{attribute 'qualified_only'}
VAR_GLOBAL CONSTANT
    nNumberOfFilterConstantThicknessSlotsInHolder : INT := 11;
    nNumberOfFilterWedgeSlotsInHolder : INT := 2;
END_VAR

(* stored: Version 1.1.0.1
   GVL PL_HE_SolidAttenuatorConstants: Id {67b56abb-a0bc-439d-804e-49b96de4219a}, ParameterList True *)
